PROGRAM prgComEffIO
VAR
	fbCom		: FB_MqttCommunicator_V5;
END_VAR

// CX-7BDACD
fbCom(
	bConnect:= TRUE, 
	strAuthKey := 'ENE87365342998',
	sUserName:= '4a0a6889-c115-4e99-9566-4029ce271fe2', 
	sUserPassword:= 'dd36787c-fc51-4107-9d6e-339f79a51c0d', 
	eSavePositionCertificate:= eSavePositionOnPLC.ePostionHardDisk,
	time_HeartBeat_sec:= T#50S, 
	bConnected=> , 
	bError=> , 
	hrErrorCode=> , 
	eConnectionState=> , 
	eErrorMessage_Out=> );

END_PROGRAM

(* stored: Version 1.1.0.1, ProductVersion 3.1.4024.15
   POU prgComEffIO: Id {cbcd318b-bf51-484c-bcaa-d6efcdf43fe3}, SpecialFunc None *)
